FUNCTION_BLOCK PICKER_VIEW_ADP_NEW_BA (* View Composite FB with adapter interface *)
  (* Standard: 61499-2 *)
  (* Version 0.2, 2003-12-05, JHC, Rockwell Automation, Renamed from NEWCOMPFB. *)
  (* Version 0.1, 2002-01-08, JHC, Rockwell Automation, Added DLY FB as example. *)
  (* Version 0.0, 2000-05-27, JHC, Rockwell Automation *)
  (* Compiler header: package fb.rt.pnp;import fb.rt.vhmi.*;import fb.rt.math.*;import fb.rt.vmath.*; *)
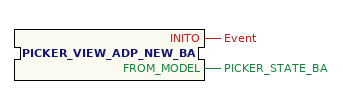
  EVENT_OUTPUT
    INITO; (* Initialization Confirm *)
  END_EVENT
  PLUGS
    FROM_MODEL : PICKER_STATE_BA;
  END_PLUGS
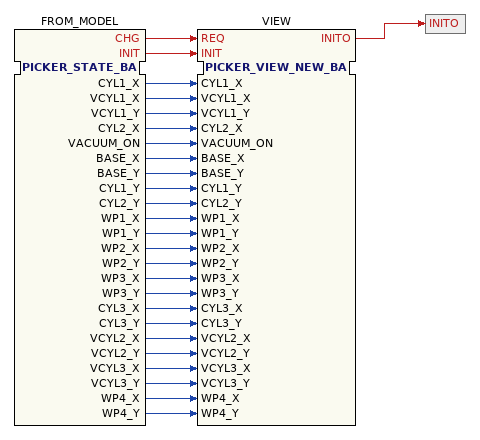
  FBS
    VIEW : PICKER_VIEW_NEW_BA;
  END_FBS
  EVENT_CONNECTIONS
    FROM_MODEL.CHG TO VIEW.REQ;
    FROM_MODEL.INIT TO VIEW.INIT;
    VIEW.INITO TO INITO;
  END_CONNECTIONS
  DATA_CONNECTIONS
    FROM_MODEL.CYL1_X TO VIEW.CYL1_X;
    FROM_MODEL.VCYL1_X TO VIEW.VCYL1_X;
    FROM_MODEL.VCYL1_Y TO VIEW.VCYL1_Y;
    FROM_MODEL.CYL2_X TO VIEW.CYL2_X;
    FROM_MODEL.VACUUM_ON TO VIEW.VACUUM_ON;
    FROM_MODEL.BASE_X TO VIEW.BASE_X;
    FROM_MODEL.BASE_Y TO VIEW.BASE_Y;
    FROM_MODEL.CYL1_Y TO VIEW.CYL1_Y;
    FROM_MODEL.CYL2_Y TO VIEW.CYL2_Y;
    FROM_MODEL.WP1_X TO VIEW.WP1_X;
    FROM_MODEL.WP1_Y TO VIEW.WP1_Y;
    FROM_MODEL.WP2_X TO VIEW.WP2_X;
    FROM_MODEL.WP2_Y TO VIEW.WP2_Y;
    FROM_MODEL.WP3_X TO VIEW.WP3_X;
    FROM_MODEL.WP3_Y TO VIEW.WP3_Y;
    FROM_MODEL.CYL3_X TO VIEW.CYL3_X;
    FROM_MODEL.CYL3_Y TO VIEW.CYL3_Y;
    FROM_MODEL.VCYL2_X TO VIEW.VCYL2_X;
    FROM_MODEL.VCYL2_Y TO VIEW.VCYL2_Y;
    FROM_MODEL.VCYL3_X TO VIEW.VCYL3_X;
    FROM_MODEL.VCYL3_Y TO VIEW.VCYL3_Y;
    FROM_MODEL.WP4_X TO VIEW.WP4_X;
    FROM_MODEL.WP4_Y TO VIEW.WP4_Y;
  END_CONNECTIONS
END_FUNCTION_BLOCK
